FUNCTION F_eVExcludeRange : DWORD
(*
    Given an lower and upper end of an exclusion range, return the corresponding eV bitmask.

    eVs between fLower and fUpper will be considered unsafe, and eVs outside of this range will be
    considered safe, with the exception of the endpoints and values near the endpoints if they land
    far from an eV boundary.

    Call this in your init cycle to set up your eV bitmasks for more readable code
    that is also more resiliant to eV range definition adjustments.
*)
VAR_INPUT
    fLower: REAL;
    fUpper: REAL;
END_VAR


F_eVExcludeRange := F_eVIncludeRange(0, fLower) OR F_eVIncludeRange(fUpper, PMPS_GVL.g_areVBoundaries[PMPS_GVL.g_cBoundaries]);

END_FUNCTION

(* stored: Version 1.1.0.1
   POU F_eVExcludeRange: Id {920777a9-efc7-465f-bdbf-e4c00c8fc260}, SpecialFunc None *)
